TYPE
    ST_IRC5_Status : STRUCT
        Extended   : BOOL;
        Retracted  : BOOL;
        Extending  : BOOL;
        Retracting : BOOL;
    END_STRUCT
END_TYPE

(* stored: Version 1.1.0.1
   DUT ST_IRC5_Status: Id {0c6cfd72-0aac-420b-9c1f-a9679b4b654d} *)
